// TIA Portal V19 export
VAR_GLOBAL   // PLC tag table "LB327"
   LB327_PareggiaturaScarico_Pb_Aux2 AT %I351.6 : Bool;   // 357SH2
   LB327_PareggiaturaScarico_Pb_Aux1 AT %I351.5 : Bool;   // 357SH1
   LB327_PareggiaturaScarico_Lp_Aux2 AT %Q351.6 : Bool;   // 357SH2
   LB327_PareggiaturaScarico_Lp_Aux1 AT %Q351.5 : Bool;   // 357SH1
END_VAR
